FUNCTION_BLOCK FB_PMLUnit IMPLEMENTS I_UnitState
VAR_INPUT
	stSubUnitInfo	: ARRAY [1..4] OF ST_PMLSubUnitInfo;	//Informations about the Subunits
END_VAR
VAR_OUTPUT
	eStateCommand	: E_PMLCommand := ePMLCommand_Abort;	//Command for a new state from superior unit
	eMode 			: DINT;
	eState 			: E_PMLState;
	bWdStatus		: BOOL;

END_VAR
VAR
fbPML_StateMachine	: PML_StateMachine;
fbPML_ModeManager	: PML_UnitModeManager;
stPackTags 			: ST_PackMLv30Ext;
rtChangeState		: R_TRIG;
rtChangeMode 		: R_TRIG;


wdState				: INT;					// Watchdog Vars
timeout 			: ARRAY [1..4] OF TON;	// Watchdog Vars
wdAlarm 			: ARRAY [1..4] OF BOOL;	// Watchdog Vars


END_VAR

fbPML_StateMachine();
fbPML_ModeManager();

// State Manager Logic
rtChangeState (CLK := stPackTags.Command.CmdChangeRequest);
	IF rtChangeState.Q THEN	
		fbPML_StateMachine.eCommand := stPackTags.Command.CntrlCmd;
	END_IF

// Mode Manager Logic	
rtChangeMode (CLK := stPackTags.Command.UnitModeChangeRequest);
	IF rtChangeMode.Q THEN
		fbPML_ModeManager.eModeCommand	:= stPackTags.Command.UnitMode;
		fbPML_ModeManager.bExecute		:= TRUE;
	END_IF
		
		IF fbPML_ModeManager.bDone THEN
			fbPML_ModeManager.bExecute := FALSE;
		END_IF
		
// Outputs to SubUnits		
eState 			:= fbPML_StateMachine.eState;	// output of local PML state
eStateCommand	:= fbPML_StateMachine.eCommand;	// output of local PML mode command
eMode			:= fbPML_StateMachine.eMode	:= fbPML_ModeManager.eModeStatus;	// output of local PML mode 

// Inputs from SubUnits
fbPML_StateMachine.stSubUnitInfoRef.ArraySize		:= SIZEOF(stSubUnitInfo);
fbPML_StateMachine.stSubUnitInfoRef.NoOfSubUnits	:= 4;
fbPML_StateMachine.stSubUnitInfoRef.pArray			:= ADR(stSubUnitInfo);

// Watchdog to monitor the PML State of the SubUnits
A_PMLWatchdog();
	bWdStatus := WdAlarm[1] OR WdAlarm[2] OR WdAlarm[3] OR WdAlarm[4];

	
// Method Calls for each PML State	
CASE eState OF
	ePMLState_Undefined:
		M_Undefined();
	ePMLState_Clearing:
		M_Clearing();
	ePMLState_Stopped:
		M_Stopped();
	ePMLState_Starting:
		M_Starting();
	ePMLState_Idle:
		M_Idle();
	ePMLState_Suspended:
		M_Suspended();
	ePMLState_Execute:
		M_Execute();
	ePMLState_Stopping:
		M_Stopping();
	ePMLState_Aborting:
		M_Aborting();
	ePMLState_Aborted:
		M_Aborted();
	ePMLState_Holding:
		M_Holding();
	ePMLState_Held:
		M_Held();
	ePMLState_Unholding:
		M_Unholding();
	ePMLState_Suspending:
		M_Suspending();
	ePMLState_Unsuspending:
		M_Unsuspending();
	ePMLState_Resetting:
		M_Resetting();
	ePMLState_Completing:
		M_Completing();
	ePMLState_Complete:
		M_Complete();
END_CASE

ACTION A_PMLWatchdog:
timeout[1](PT:= T#7S);
timeout[2](PT:= T#7S);
timeout[3](PT:= T#7S);
timeout[4](PT:= T#7S);


CASE wdState OF
	
	0:
		IF stSubUnitInfo[1].Active THEN
			timeout[1].IN	:= TRUE;
			wdState			:= 5;
		ELSE
			wdState			:= 10;	
		END_IF
	5:
		IF stSubUnitInfo[1].eState = eState THEN
			wdAlarm[1]		:= FALSE;
			timeout[1].IN	:= FALSE;
			wdState			:= 10;
		ELSIF timeout[1].Q THEN
			wdAlarm[1]		:= TRUE;
			timeout[1].IN	:= FALSE;
			wdState			:= 10;
		END_IF
	10:
		IF stSubUnitInfo[2].Active THEN
			timeout[2].IN	:= TRUE;
			wdState			:= 15;
		ELSE
			wdState			:= 20;	
		END_IF
	15:
		IF stSubUnitInfo[2].eState = eState THEN
			wdAlarm[2]		:= FALSE;
			timeout[2].IN	:= FALSE;
			wdState			:= 20;
		ELSIF timeout[2].Q THEN
			wdAlarm[2]		:= TRUE;
			timeout[2].IN	:= FALSE;
			wdState			:= 20;
		END_IF
	20:
		IF stSubUnitInfo[3].Active THEN
			timeout[3].IN	:= TRUE;
			wdState			:= 25;
		ELSE
			wdState			:= 30;
		END_IF
	25:
		IF stSubUnitInfo[3].eState = eState THEN
			wdAlarm[3]		:= FALSE;
			timeout[3].IN	:= FALSE;
			wdState			:= 30;
		ELSIF timeout[3].Q THEN
			wdAlarm[3]		:= TRUE;
			timeout[3].IN	:= FALSE;
			wdState			:= 30;
		END_IF
	30:
		IF stSubUnitInfo[4].Active THEN
			timeout[4].IN	:= TRUE;
			wdState			:= 35;
		ELSE
			wdState			:= 0;
		END_IF
	35:
		IF stSubUnitInfo[4].eState = eState THEN
			wdAlarm[4]		:= FALSE;
			timeout[4].IN	:= FALSE;
			wdState			:= 0;
		ELSIF timeout[4].Q THEN
			wdAlarm[4]		:= TRUE;
			timeout[4].IN	:= FALSE;
			wdState			:= 0;
		END_IF	
		
END_CASE
END_ACTION

{warning 'add method implementation '}
METHOD M_Aborted
END_METHOD

{warning 'add method implementation '}
METHOD M_Aborting
M_StateComplete();
END_METHOD

{warning 'add method implementation '}
METHOD M_Clearing
M_StateComplete();
END_METHOD

{warning 'add method implementation '}
METHOD M_Complete
END_METHOD

{warning 'add method implementation '}
METHOD M_Completing
M_StateComplete();
END_METHOD

{warning 'add method implementation '}
METHOD M_Execute
END_METHOD

{warning 'add method implementation '}
METHOD M_Held
END_METHOD

{warning 'add method implementation '}
METHOD M_Holding
M_StateComplete();
END_METHOD

{warning 'add method implementation '}
METHOD M_Idle
END_METHOD

{warning 'add method implementation '}
METHOD M_Resetting
M_StateComplete();
END_METHOD

{warning 'add method implementation '}
METHOD M_Starting
M_StateComplete();
END_METHOD

{warning 'add method implementation '}
METHOD M_StateComplete
fbPML_StateMachine.M_StateComplete();
END_METHOD

{warning 'add method implementation '}
METHOD M_Stopped
END_METHOD

{warning 'add method implementation '}
METHOD M_Stopping
M_StateComplete();
END_METHOD

{warning 'add method implementation '}
METHOD M_Suspended
M_StateComplete();
END_METHOD

{warning 'add method implementation '}
METHOD M_Suspending
M_StateComplete();
END_METHOD

{warning 'add method implementation '}
METHOD M_Undefined
END_METHOD

{warning 'add method implementation '}
METHOD M_Unholding
END_METHOD

{warning 'add method implementation '}
METHOD M_Unsuspending
END_METHOD

PROPERTY P_PackTags : REFERENCE TO ST_PackMLv30Ext
GET
P_PackTags REF= stPackTags;
END_GET
SET
stPackTags := P_PackTags;
END_SET
END_PROPERTY

END_FUNCTION_BLOCK

(* stored: Version 1.1.0.1, ProductVersion 3.1.4024.11
   POU FB_PMLUnit: Id {76d81add-3ba6-490e-91ea-f5b930ee47b5}, SpecialFunc None
   Folder Pack Tags: Id {328ed5ed-6360-4bb7-8672-1ad4c0a7ef7e}
   Folder PML States: Id {5b089b78-2d2a-467f-9757-b140acb3b63d}
   Action A_PMLWatchdog: Id {8ac386db-4cf3-420f-9f5a-f6ffde21fe88}
   Method M_Aborted: Id {fba60604-4588-400d-91a9-dd653bcbf5d0}
   Method M_Aborting: Id {d6ba3c67-8fba-46c9-a5d0-b49d7852c9de}
   Method M_Clearing: Id {23f6b7f4-b18a-4812-8a92-218b357f5daf}
   Method M_Complete: Id {97527de1-1ae8-4069-8fb8-c9c8d0501ac8}
   Method M_Completing: Id {294a2300-f39d-4b55-8788-6d4ce03d70dc}
   Method M_Execute: Id {b824c714-1c4c-4058-b256-fb25750fe1d4}
   Method M_Held: Id {61d0b5bd-d88d-46cc-81dd-b5df83b3ec1f}
   Method M_Holding: Id {1af8cb2b-36ac-461d-b019-af3df1ab8634}
   Method M_Idle: Id {aef35c11-f5f1-40d6-9ee2-b9df3b4388a1}
   Method M_Resetting: Id {6ec0d892-db77-427c-8e90-7274bf7d178e}
   Method M_Starting: Id {b9ed8a13-a400-4b6c-b112-4f0ec389b84e}
   Method M_StateComplete: Id {5468dcf1-3449-4fee-8be2-b88f8d1de6ce}
   Method M_Stopped: Id {154c7d10-3861-4016-8b90-fde1b202d946}
   Method M_Stopping: Id {7432c237-396b-4548-b68d-b6955721e05f}
   Method M_Suspended: Id {fd0f4230-a78b-4ed1-8cf6-e8cd9c86044f}
   Method M_Suspending: Id {a57884f9-4a0c-466c-88b7-08ba1a5cbecc}
   Method M_Undefined: Id {c4144a95-7feb-4cd6-a703-d3f7d7af6ed2}
   Method M_Unholding: Id {9dd0a3d1-f78c-4255-882d-3fbc253e2566}
   Method M_Unsuspending: Id {7c02729b-973f-43dd-bc27-931fea9ae236}
   Property P_PackTags: Id {d4fd7f25-fac9-4d63-97d8-fd9490de3af8}
   Get Get: Id {defbd6b3-564a-47bb-94ea-5385093654d3}
   Set Set: Id {79c99a0d-6a60-4afd-badd-09c0eaef16fd} *)
